// TIA Portal V20 export
DATA_BLOCK "IF_HMI_FB_IDB"   // DB30222
// stored: AutoNumber false, InstanceOfName IF_HMI_FB, InstanceOfType FB
"IF_HMI_FB"
   // VAR_INPUT
   //    INIT_HMI_OPMODE { ExternalAccessible := 'False'; ExternalVisible := 'False'; ExternalWritable := 'False'} : "INIT_HMI_OPMODE_UDT";
   //    CLOCK_SYSTEM_INFO : "GLOBAL_CLOCK&SYSTEM_MEMORY_UDT";
   // END_VAR
   // VAR_IN_OUT
   //    OPERATOR_PROMPT_IF : "OPERATOR_PROMPT_UDT";
   // END_VAR
   // VAR
   //    "IF" { S7_SetPoint := 'True'} : "IF_HMI_UDT";
   //    "RT_INFO.INFO" { ExternalAccessible := 'False'; ExternalVisible := 'False'; ExternalWritable := 'False'} : LTime;
   //    "RT_INFO.RET_VAL" { ExternalAccessible := 'False'; ExternalVisible := 'False'; ExternalWritable := 'False'} : Word;
   //    CycleConvert { ExternalAccessible := 'False'; ExternalVisible := 'False'; ExternalWritable := 'False'} : Int;
   //    LimitValue { ExternalAccessible := 'False'; ExternalVisible := 'False'; ExternalWritable := 'False'} : Int;
   // END_VAR
BEGIN
END_DATA_BLOCK
